PROGRAM MAIN
VAR
	/// axis reference data structure 
	Axis1: AXIS_REF;
END_VAR

METHOD ShiftRegister
VAR
	fbPulse : FB_PulseGenerate2s;	
	
	bStart: BOOL;
	
    nInByte  :  BYTE:=16#01; (*2#0100 0101*)   
    nVar : BYTE  := 1; 
	
	rt : R_TRIG;
	bSensor: BOOL;
	rtSensor : R_TRIG;
	
	rtCam1:R_TRIG;
	bCam1 : UINT;
END_VAR
fbPulse(bExcute:=bStart);

rt(CLK:=fbPulse.Q);
IF rt.Q THEN
	nInByte := SHL(nInByte,nVar);
END_IF

//register point
rtSensor(CLK:=bSensor);
IF rtSensor.Q THEN
	bSensor:= FALSE;
	nInByte := nInByte OR 16#01;
END_IF
//get bit at 9th position
rtCam1(CLK:=nInByte.3);
IF rtCam1.Q THEN
	bCam1:=bCam1+1;
END_IF
END_METHOD

END_PROGRAM

(* stored: Version 1.1.0.1, ProductVersion 3.1.4024.12
   POU MAIN: Id {de2cbbea-be5d-40b1-a141-edaf4becbde4}, SpecialFunc None
   Method ShiftRegister: Id {ac29a83c-8972-4d3b-8a3a-f827c81d81d1} *)
